INTERFACE IStepManager
// Copyright (c) 2024 Loupe (https://loupe.team), provided under the MIT License.

METHOD _requestStep : BOOL
VAR_INPUT
	nextStep : ENUM;
END_VAR
END_METHOD

METHOD _reset : BOOL
VAR_INPUT
END_VAR
END_METHOD

METHOD _sequenceComplete : BOOL
VAR_INPUT
END_VAR
END_METHOD

METHOD _sequenceError : BOOL
VAR_INPUT
END_VAR
END_METHOD

PROPERTY currentStep : ENUM
GET
END_GET
END_PROPERTY

PROPERTY RequestNumber : DINT
GET
END_GET
END_PROPERTY

END_INTERFACE

(* stored: Version 1.1.0.1
   Itf IStepManager: Id {89c191eb-450f-4144-a19d-873d9f6fc237}
   Method _requestStep: Id {484e6cd7-60ba-4268-b695-64585da66145}
   Method _reset: Id {c44b696d-696b-4673-a947-9ec390e7c67e}
   Method _sequenceComplete: Id {f41bcaea-5de9-45b2-807e-ba3bb516ac9c}
   Method _sequenceError: Id {346d84e2-d277-4231-a765-0b63457bf8e8}
   Property currentStep: Id {f549aba3-dc6c-45db-ae21-2b43a54633f2}
   Get Get: Id {e53bfbc9-86ad-48ac-b648-09cfbdc36fb7}
   Property RequestNumber: Id {48610b89-952c-4a85-87b0-3a800ad674d5}
   Get Get: Id {562ca9eb-e252-47f1-9d0d-9ab9f5f5f405} *)
